// TIA Portal project "Motor_VFD" (V15.1)

(* hardware
DEVICE "S71500/ET200MP station_1"  S7-1500 station
   slot 0: "Rail_0"  Rack  6ES7 590-1***0-0AA0
   slot 1: "PLC_1"  CPU 1513-1 PN  6ES7 513-1AL02-0AB0  V2.6
      slot 3: "CPU display_1"  6ES7591-1AA00-0AA0
DEVICE "HMI_1"  KTP900 Basic PN
   slot 0: "HMI_1"  KTP900 Basic PN  6AV2 123-2JB03-0AX0  15.1.0.0
   slot 1: "HMI_RT_1"  KTP900 Basic PN  6AV2 123-2JB03-0AX0  15.1.0.0
   slot 5: "HMI_1.IE_CP_1"  PROFINET Interface  15.0.1.0
      slot 1: "PROFINET Interface_1"  PROFINET Interface
         slot 1: "Port_1"  Port
*)

// ===== PLC "PLC_1"  CPU 1513-1 PN =====

VAR_GLOBAL   // PLC tag table "Default tag table"
   "Clock_Byte" AT %MB8080 : Byte;
   "Clock_10Hz" AT %M8080.0 : Bool;
   "Clock_5Hz" AT %M8080.1 : Bool;
   "Clock_2.5Hz" AT %M8080.2 : Bool;
   "Clock_2Hz" AT %M8080.3 : Bool;
   "Clock_1.25Hz" AT %M8080.4 : Bool;
   "Clock_1Hz" AT %M8080.5 : Bool;
   "Clock_0.625Hz" AT %M8080.6 : Bool;
   "Clock_0.5Hz" AT %M8080.7 : Bool;
END_VAR

// folder: Instante

DATA_BLOCK "SoftStarter_DB"   // DB3
{ S7_Optimized_Access := 'TRUE' }
VERSION : 0.1
// stored: InstanceOfName SoftStarter
"SoftStarter"
BEGIN
END_DATA_BLOCK

DATA_BLOCK "VFD_DB"   // DB4
{ S7_Optimized_Access := 'TRUE' }
VERSION : 0.1
// stored: InstanceOfName VFD
"VFD"
BEGIN
END_DATA_BLOCK

// folder: SoftStart

DATA_BLOCK "SoftStarter_DB_Motor"   // DB1
{ S7_Optimized_Access := 'TRUE' }
VERSION : 0.1
   VAR
      start : Bool;
      stop : Bool;
      running : Bool;
      bypassed : Bool;
      rampUpTime : Real := 10.0;
      rampDownTime : Real := 5.0;
      startVoltagePct : Real := 30.0;
      fullLoadAmp : Real := 50.0;
      motorRatedRPM : Real := 1450.0;
      motorSpeed : Real;
      motorCurrent : Real;
      actualVoltagePct : Real;
      state : Int;
   END_VAR
BEGIN
END_DATA_BLOCK

// folder: VFD

DATA_BLOCK "VFD_DB_Motor"   // DB2
{ S7_Optimized_Access := 'TRUE' }
VERSION : 0.1
   VAR
      enable : Bool;
      ready : Bool;
      running : Bool;
      atSetpoint : Bool;
      actualFreqHz : Real;
      motorSpeed : Real;
      motorCurrent : Real;
      speedSetpointHz : Real;
      accelTime : Real := 10.0;
      decel_time : Real := 10.0;
      maxFreqHz : Real := 50.0;
      fullLoadAmps : Real := 50.0;
      motorRatedRPM : Real := 1450.0;
   END_VAR
BEGIN
END_DATA_BLOCK

// folder: (top level)

ORGANIZATION_BLOCK "Main"   // OB1, LAD, ProgramCycle
TITLE = "Main Program Sweep (Cycle)"
{ S7_Optimized_Access := 'TRUE' }
VERSION : 0.1
   VAR_INPUT
      Initial_Call : Bool;   // Initial call of this OB
      Remanence : Bool;   // =True, if remanent data are available
   END_VAR
BEGIN
END_ORGANIZATION_BLOCK

ORGANIZATION_BLOCK "Simulare"   // OB30, LAD, CyclicInterrupt
{ S7_Optimized_Access := 'TRUE' }
VERSION : 0.1
   VAR_INPUT
      Initial_Call : Bool;   // Initial call of this OB
      Event_Count : Int;   // Events discarded
   END_VAR
BEGIN

REGION Network 1: Soft Starter
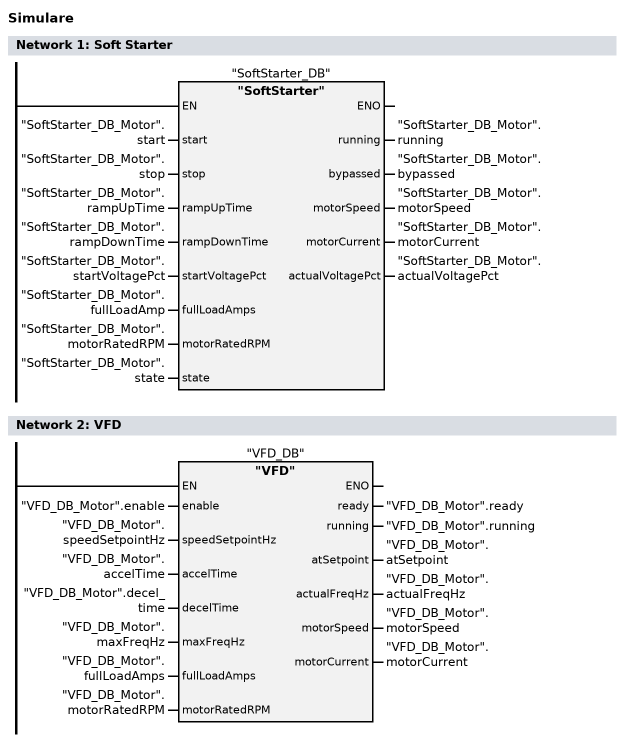
   RUNG wire#powerrail
      "SoftStarter_DB"(start := "SoftStarter_DB_Motor".start, stop := "SoftStarter_DB_Motor".stop, rampUpTime := "SoftStarter_DB_Motor".rampUpTime, rampDownTime := "SoftStarter_DB_Motor".rampDownTime, startVoltagePct := "SoftStarter_DB_Motor".startVoltagePct, fullLoadAmps := "SoftStarter_DB_Motor".fullLoadAmp, motorRatedRPM := "SoftStarter_DB_Motor".motorRatedRPM, state := "SoftStarter_DB_Motor".state, running => "SoftStarter_DB_Motor".running, bypassed => "SoftStarter_DB_Motor".bypassed, motorSpeed => "SoftStarter_DB_Motor".motorSpeed, motorCurrent => "SoftStarter_DB_Motor".motorCurrent, actualVoltagePct => "SoftStarter_DB_Motor".actualVoltagePct)
   END_RUNG
   // the same network as SCL:
   "SoftStarter_DB"(start := "SoftStarter_DB_Motor".start,   // "SoftStarter"
                    stop := "SoftStarter_DB_Motor".stop,
                    rampUpTime := "SoftStarter_DB_Motor".rampUpTime,
                    rampDownTime := "SoftStarter_DB_Motor".rampDownTime,
                    startVoltagePct := "SoftStarter_DB_Motor".startVoltagePct,
                    fullLoadAmps := "SoftStarter_DB_Motor".fullLoadAmp,
                    motorRatedRPM := "SoftStarter_DB_Motor".motorRatedRPM,
                    state := "SoftStarter_DB_Motor".state,
                    running => "SoftStarter_DB_Motor".running,
                    bypassed => "SoftStarter_DB_Motor".bypassed,
                    motorSpeed => "SoftStarter_DB_Motor".motorSpeed,
                    motorCurrent => "SoftStarter_DB_Motor".motorCurrent,
                    actualVoltagePct => "SoftStarter_DB_Motor".actualVoltagePct);
END_REGION

REGION Network 2: VFD
   RUNG wire#powerrail
      "VFD_DB"(enable := "VFD_DB_Motor".enable, speedSetpointHz := "VFD_DB_Motor".speedSetpointHz, accelTime := "VFD_DB_Motor".accelTime, decelTime := "VFD_DB_Motor".decel_time, maxFreqHz := "VFD_DB_Motor".maxFreqHz, fullLoadAmps := "VFD_DB_Motor".fullLoadAmps, motorRatedRPM := "VFD_DB_Motor".motorRatedRPM, ready => "VFD_DB_Motor".ready, running => "VFD_DB_Motor".running, atSetpoint => "VFD_DB_Motor".atSetpoint, actualFreqHz => "VFD_DB_Motor".actualFreqHz, motorSpeed => "VFD_DB_Motor".motorSpeed, motorCurrent => "VFD_DB_Motor".motorCurrent)
   END_RUNG
   // the same network as SCL:
   "VFD_DB"(enable := "VFD_DB_Motor".enable,   // "VFD"
            speedSetpointHz := "VFD_DB_Motor".speedSetpointHz,
            accelTime := "VFD_DB_Motor".accelTime,
            decelTime := "VFD_DB_Motor".decel_time,
            maxFreqHz := "VFD_DB_Motor".maxFreqHz,
            fullLoadAmps := "VFD_DB_Motor".fullLoadAmps,
            motorRatedRPM := "VFD_DB_Motor".motorRatedRPM,
            ready => "VFD_DB_Motor".ready,
            running => "VFD_DB_Motor".running,
            atSetpoint => "VFD_DB_Motor".atSetpoint,
            actualFreqHz => "VFD_DB_Motor".actualFreqHz,
            motorSpeed => "VFD_DB_Motor".motorSpeed,
            motorCurrent => "VFD_DB_Motor".motorCurrent);
END_REGION
END_ORGANIZATION_BLOCK

// folder: SoftStart

FUNCTION_BLOCK "SoftStarter"   // FB1, SCL
{ S7_Optimized_Access := 'TRUE' }
VERSION : 0.1
   VAR_INPUT
      start : Bool;
      stop : Bool;
      rampUpTime : Real := 0.0;
      rampDownTime : Real := 0.0;
      startVoltagePct : Real := 0.0;
      fullLoadAmps : Real := 0.0;
      motorRatedRPM : Real := 0.0;
   END_VAR
   VAR_OUTPUT
      running : Bool;
      bypassed : Bool;
      motorSpeed : Real;
      motorCurrent : Real;
      actualVoltagePct : Real;
   END_VAR
   VAR_IN_OUT
      state : Int;
   END_VAR
   VAR
      timerAcc : Real;
   END_VAR
BEGIN
   IF #stop THEN
       IF #state = 1 OR #state = 2 THEN
           #state := 3; // Force Ramp Down
           #timerAcc := 0.0;
       END_IF;
   END_IF;

   CASE #state OF
       0: //oprit
           #actualVoltagePct := 0.0;
           #motorSpeed := 0.0;
           #motorCurrent := 0.0;
           #running := FALSE;
           #bypassed := FALSE;
           #timerAcc := 0.0;

           IF #start AND NOT #stop THEN
               #state := 1; //incepe pe ramp up
           END_IF;
       1: //ramp up
           #running := TRUE;
           #bypassed := FALSE;
           #timerAcc := #timerAcc + 0.1;

           //rampa liniara de tensiune de la #startVoltagePct la 100%
           IF #rampUpTime > 0.0 THEN
               #actualVoltagePct := #startVoltagePct + ((100.0 - #startVoltagePct) * (#timerAcc / #rampUpTime));
           ELSE
               #actualVoltagePct := 100.0;
           END_IF;

           IF #actualVoltagePct > 100.0 THEN
               #actualVoltagePct := 100.0;
           END_IF;

           //viteza urmareste rampa de tensiune non-linear
           #motorSpeed := #motorRatedRPM * (#actualVoltagePct / 100.0);

           //curentul de pornire ramane ridicat pana ajunge la viteza maxima
           #motorCurrent := #fullLoadAmps * 3.5 * (#actualVoltagePct / 100.0);

           IF #actualVoltagePct >= 100.0 OR #timerAcc >= #rampUpTime THEN
               #actualVoltagePct := 100.0;
               #state := 2;
               #timerAcc := 0.0;
           END_IF;
       2: //bypas (viteza maxima)
           #running := TRUE;
           #bypassed := TRUE;
           #actualVoltagePct := 100.0;
           #motorSpeed := #motorRatedRPM;
           #motorCurrent := #fullLoadAmps; //curent normal pe motor

           IF #stop THEN
               #state := 3;
               #timerAcc := 0.0;
           END_IF;
       3: //ramp down pentru oprire motor
           #bypassed := FALSE;
           #timerAcc := #timerAcc + 0.1;

           IF #rampDownTime > 0.0 THEN
               #actualVoltagePct := 100.0 - ((100.0 - #startVoltagePct) * (#timerAcc / #rampDownTime));
           ELSE
               #actualVoltagePct := 0.0;
           END_IF;

           #motorSpeed := #motorRatedRPM * (#actualVoltagePct / 100.0);
           #motorCurrent := #fullLoadAmps * (#actualVoltagePct / 100.0);

           IF #actualVoltagePct <= #startVoltagePct OR #timerAcc >= #rampDownTime THEN
               #state := 0;
           END_IF;
   END_CASE;
END_FUNCTION_BLOCK

// folder: VFD

FUNCTION_BLOCK "VFD"   // FB2, SCL
{ S7_Optimized_Access := 'TRUE' }
VERSION : 0.1
   VAR_INPUT
      enable : Bool;
      speedSetpointHz : Real;
      accelTime : Real := 10.0;
      decelTime : Real := 10.0;
      maxFreqHz : Real := 50.0;
      fullLoadAmps : Real := 50.0;
      motorRatedRPM : Real := 1450.0;
   END_VAR
   VAR_OUTPUT
      ready : Bool;
      running : Bool;
      atSetpoint : Bool;
      actualFreqHz : Real;
      motorSpeed : Real;
      motorCurrent : Real;
   END_VAR
   VAR
      cycleTimeSec : Real := 0.1;
   END_VAR
BEGIN
   #ready := TRUE;

   IF #enable THEN
       #running := TRUE;

       //calcul pentru frecventa maxima per pas pentru cicluri de 0.1s
       // pas = (frecventaMAxima / timpDeRampa) * timpCiclu
       IF #actualFreqHz < #speedSetpointHz THEN
           //accelereaza
           IF #accelTime > 0.0 THEN
               #actualFreqHz := #actualFreqHz + ((#maxFreqHz / #accelTime) * 0.1);
           ELSE
               #actualFreqHz := #speedSetpointHz;
           END_IF;

           IF #actualFreqHz > #speedSetpointHz THEN
               #actualFreqHz := #speedSetpointHz;
           END_IF;

           //curentul la accelerare = cuentul de magnetizare(30%) + curentul de cuplu(120%) 
           #motorCurrent := #fullLoadAmps * 1.2;
       ELSIF #actualFreqHz > #speedSetpointHz THEN
           //decelereaza
           IF #decelTime > 0.0 THEN
               #actualFreqHz := #actualFreqHz - ((#maxFreqHz / #decelTime) * 0.1);
           ELSE
               #actualFreqHz := #speedSetpointHz;
           END_IF;

           IF #actualFreqHz < #speedSetpointHz THEN
               #actualFreqHz := #speedSetpointHz;
           END_IF;

           #motorCurrent := #fullLoadAmps * 0.8;
       ELSE //echilibru (steay state) la setpoint
           #motorCurrent := #fullLoadAmps * (#actualFreqHz / #maxFreqHz);
       END_IF;

       //flag pentru statusul la iesire
       #atSetpoint := (ABS(#actualFreqHz - #speedSetpointHz) < 0.1);

       //outpul la viteza proportional: viteza = (freq / maxFreq) * rateRPM
       #motorSpeed := (#actualFreqHz / #maxFreqHz) * #motorRatedRPM;

   ELSE
       //decelereaza la zero
       #atSetpoint := FALSE;
       IF #actualFreqHz > 0.0 THEN
           #actualFreqHz := #actualFreqHz - ((#maxFreqHz / #decelTime) * 0.1);
           IF #actualFreqHz < 0.0 THEN
               #actualFreqHz := 0.0;
           END_IF;
           #motorSpeed := (#actualFreqHz / #maxFreqHz) * #motorRatedRPM;
           #motorCurrent := #fullLoadAmps * 0.3; //curent rezidual
       ELSE
           #actualFreqHz := 0.0;
           #motorSpeed := 0.0;
           #motorCurrent := 0.0;
           #running := FALSE;
       END_IF;
   END_IF;
END_FUNCTION_BLOCK

(* ===== HMI "HMI_RT_1" =====
system functions are stored by id; their names below are inferred from use
connection "HMI_Connection_1": ETHERNET, SMART_S7_1500_OMS

HMI tags "Default tag table"
   "SoftStarter_DB_Motor_state" : Int = PLC SoftStarter_DB_Motor.state, 1 s
   "SoftStarter_DB_Motor_start" : Bool = PLC SoftStarter_DB_Motor.start, 1 s
   "SoftStarter_DB_Motor_stop" : Bool = PLC SoftStarter_DB_Motor.stop, 1 s
   "SoftStarter_DB_Motor_rampUpTime" : Real = PLC SoftStarter_DB_Motor.rampUpTime, 1 s
   "SoftStarter_DB_Motor_rampDownTime" : Real = PLC SoftStarter_DB_Motor.rampDownTime, 1 s
   "SoftStarter_DB_Motor_startVoltagePct" : Real = PLC SoftStarter_DB_Motor.startVoltagePct, 1 s
   "SoftStarter_DB_Motor_fullLoadAmp" : Real = PLC SoftStarter_DB_Motor.fullLoadAmp, 1 s
   "SoftStarter_DB_Motor_motorRatedRPM" : Real = PLC SoftStarter_DB_Motor.motorRatedRPM, 1 s
   "SoftStarter_DB_Motor_motorSpeed" : Real = PLC SoftStarter_DB_Motor.motorSpeed, 1 s
   "SoftStarter_DB_Motor_motorCurrent" : Real = PLC SoftStarter_DB_Motor.motorCurrent, 1 s
   "SoftStarter_DB_Motor_actualVoltagePct" : Real = PLC SoftStarter_DB_Motor.actualVoltagePct, 1 s
   "VFD_DB_Motor_enable" : Bool = PLC VFD_DB_Motor.enable, 1 s
   "VFD_DB_Motor_speedSetpointHz" : Real = PLC VFD_DB_Motor.speedSetpointHz, 1 s
   "VFD_DB_Motor_accelTime" : Real = PLC VFD_DB_Motor.accelTime, 1 s
   "VFD_DB_Motor_decel_time" : Real = PLC VFD_DB_Motor.decel_time, 1 s
   "VFD_DB_Motor_maxFreqHz" : Real = PLC VFD_DB_Motor.maxFreqHz, 1 s
   "VFD_DB_Motor_fullLoadAmps" : Real = PLC VFD_DB_Motor.fullLoadAmps, 1 s
   "VFD_DB_Motor_motorRatedRPM" : Real = PLC VFD_DB_Motor.motorRatedRPM, 1 s
   "VFD_DB_Motor_running" : Bool = PLC VFD_DB_Motor.running, 1 s
   "VFD_DB_Motor_atSetpoint" : Bool = PLC VFD_DB_Motor.atSetpoint, 1 s
   "VFD_DB_Motor_actualFreqHz" : Real = PLC VFD_DB_Motor.actualFreqHz, 1 s
   "VFD_DB_Motor_motorSpeed" : Real = PLC VFD_DB_Motor.motorSpeed, 1 s
   "VFD_DB_Motor_motorCurrent" : Real = PLC VFD_DB_Motor.motorCurrent, 1 s

screen "VFD" 800x480, template "Template_1"
   TextField "Text field_1" at 36,447 size 29x20; Text 'VFD'
   TextField "Text field_2" at 118,447 size 70x20; Text 'Soft Start'
   TextField "Text field_3" at 382,15 size 51x32; Text 'VFD'
   GraphicView "Graphic view_2" at 281,151 size 276x171; Picture "Graphic_3"
   GraphicView "Graphic view_4" at 281,151 size 276x171; Picture "Graphic_7"
      Visibility <- "VFD_DB_Motor_running"
   GraphicView "Graphic view_1" at 281,151 size 276x171; Picture "Graphic_6"
      Visibility <- "VFD_DB_Motor_atSetpoint"
   Button "Button_1" at 235,193 size 52x32; TextOff 'Start'
      on Press: SetBit("VFD_DB_Motor_enable")
   Button "Button_2" at 235,225 size 52x32; TextOff 'Stop'
      on Press: ResetBit("VFD_DB_Motor_enable")
   TextField "Text field_4" at 53,14 size 104x25; Text 'Valori input'
   TextField "Text field_5" at 14,76 size 133x20; Text 'Setpoint frecventa:'
   TextField "Text field_6" at 12,155 size 113x20; Text 'Timp decelerare:'
   TextField "Text field_7" at 13,195 size 105x20; Text 'Frecventa max:'
   TextField "Text field_8" at 14,240 size 107x20; Text 'Curent nominal:'
   TextField "Text field_15" at 15,288 size 91x20; Text 'RPM nominal:'
   IOField "I/O field_1" at 149,74 size 42x26; FormatPattern 99.9
      ProcessValue <- "VFD_DB_Motor_speedSetpointHz"
   IOField "I/O field_7" at 128,153 size 42x26; FormatPattern 99.9
      ProcessValue <- "VFD_DB_Motor_decel_time"
   IOField "I/O field_8" at 120,193 size 46x26; FormatPattern 99.9
      ProcessValue <- "VFD_DB_Motor_maxFreqHz"
   IOField "I/O field_9" at 123,238 size 43x26; FormatPattern 99.9
      ProcessValue <- "VFD_DB_Motor_fullLoadAmps"
   IOField "I/O field_10" at 108,285 size 58x26; FormatPattern 9999.9
      ProcessValue <- "VFD_DB_Motor_motorRatedRPM"
   TextField "Text field_9" at 12,114 size 112x20; Text 'Timp accelerare:'
   IOField "I/O field_2" at 128,112 size 42x26; FormatPattern 99.9
      ProcessValue <- "VFD_DB_Motor_accelTime"
   TextField "Text field_10" at 638,282 size 117x25; Text 'Valori output'
   TextField "Text field_19" at 607,391 size 94x20; Text 'Viteza motor:'
   TextField "Text field_20" at 608,343 size 127x20; Text 'Frecventa actuala:'
   IOField "I/O field_4" at 706,389 size 60x26; FormatPattern 9999.9
      ProcessValue <- "VFD_DB_Motor_motorSpeed"
   IOField "I/O field_11" at 736,340 size 44x26; FormatPattern 99.9
      ProcessValue <- "VFD_DB_Motor_actualFreqHz"
   TextField "Text field_11" at 607,436 size 97x20; Text 'Curent motor:'
   IOField "I/O field_3" at 708,434 size 53x26; FormatPattern 999.9
      ProcessValue <- "VFD_DB_Motor_motorCurrent"

screen "SoftStarter" 800x480
   TextField "Text field_1" at 36,447 size 29x20; Text 'VFD'
   TextField "Text field_2" at 118,447 size 70x20; Text 'Soft Start'
   TextField "Text field_3" at 348,14 size 119x32; Text 'Soft Start'
   GraphicView "Graphic view_2" at 281,151 size 276x171; Picture "Graphic_3"
      Visibility <- "SoftStarter_DB_Motor_state"
   GraphicView "Graphic view_1" at 281,152 size 276x171; Picture "Graphic_6"
      Visibility <- "SoftStarter_DB_Motor_state"
   GraphicView "Graphic view_3" at 281,152 size 276x171; Picture "Graphic_7"
      Visibility <- "SoftStarter_DB_Motor_state"
   GraphicView "Graphic view_4" at 281,152 size 276x171; Picture "Graphic_7"
      Visibility <- "SoftStarter_DB_Motor_state"
   IOField "I/O field_1" at 424,125 size 20x20; FormatPattern 9
      ProcessValue <- "SoftStarter_DB_Motor_state"
   TextField "Text field_4" at 374,123 size 51x22; Text 'Stare:'
   TextField "Text field_5" at 617,31 size 109x20; Text 'Stari: 0 -> oprit'
   TextField "Text field_6" at 657,47 size 85x20; Text '1 -> pornire'
   TextField "Text field_7" at 657,63 size 84x20; Text '2 -> bypass'
   TextField "Text field_8" at 658,79 size 77x20; Text '3 -> oprire'
   Button "Button_1" at 235,193 size 52x32; TextOff 'Start'
      on Press: SetBit("SoftStarter_DB_Motor_start")
      on Release: ResetBit("SoftStarter_DB_Motor_start")
   Button "Button_2" at 235,225 size 52x32; TextOff 'Stop'
      on Press: SetBit("SoftStarter_DB_Motor_stop")
      on Release: ResetBit("SoftStarter_DB_Motor_stop")
   TextField "Text field_9" at 53,14 size 104x25; Text 'Valori input'
   TextField "Text field_10" at 14,76 size 90x20; Text 'Timp pornire:'
   TextField "Text field_11" at 14,127 size 82x20; Text 'Timp oprire:'
   TextField "Text field_12" at 13,176 size 104x20; Text 'Tensiune start:'
   TextField "Text field_13" at 14,221 size 107x20; Text 'Curent nominal:'
   TextField "Text field_14" at 15,269 size 91x20; Text 'RPM nominal:'
   IOField "I/O field_2" at 108,75 size 42x26; FormatPattern 99.9
      ProcessValue <- "SoftStarter_DB_Motor_rampUpTime"
   IOField "I/O field_3" at 99,125 size 42x26; FormatPattern 99.9
      ProcessValue <- "SoftStarter_DB_Motor_rampDownTime"
   IOField "I/O field_4" at 120,174 size 56x26; FormatPattern 99.9; Unit %
      ProcessValue <- "SoftStarter_DB_Motor_startVoltagePct"
   IOField "I/O field_5" at 123,219 size 43x26; FormatPattern 99.9
      ProcessValue <- "SoftStarter_DB_Motor_fullLoadAmp"
   IOField "I/O field_6" at 108,266 size 58x26; FormatPattern 9999.9
      ProcessValue <- "SoftStarter_DB_Motor_motorRatedRPM"
   TextField "Text field_15" at 638,282 size 117x25; Text 'Valori output'
   TextField "Text field_18" at 606,438 size 110x20; Text 'Tensiune motor:'
   TextField "Text field_19" at 607,391 size 97x20; Text 'Curent motor:'
   TextField "Text field_20" at 608,343 size 99x20; Text 'Turatie motor:'
   IOField "I/O field_7" at 720,436 size 65x26; FormatPattern 999.9; Unit %
      ProcessValue <- "SoftStarter_DB_Motor_actualVoltagePct"
   IOField "I/O field_8" at 708,389 size 53x26; FormatPattern 999.9
      ProcessValue <- "SoftStarter_DB_Motor_motorCurrent"
   IOField "I/O field_11" at 710,340 size 58x26; FormatPattern 9999.9
      ProcessValue <- "SoftStarter_DB_Motor_motorSpeed"
*)